// TIA Portal V16 export
// export: Created 2024-03-27T10:00:42.5235415Z, ExportSetting WithDefaults, DisplayName Totally Integrated Automation Portal, DisplayVersion V16, DisplayName TIA Portal Version Control Interface, DisplayVersion V16, DisplayName TIA Portal Openness, DisplayVersion V16, DisplayName STEP 7 Professional, DisplayVersion V16, DisplayName STEP 7 Safety, DisplayVersion V16, DisplayName WinCC Advanced, DisplayVersion V16
TYPE "UR_1_T2O_State"
// stored: IsFailsafeCompliant false
   STRUCT
      Robot { S7_SetPoint := 'True'} : "UR__T2O_Robot";
      Safety { S7_SetPoint := 'True'} : "UR__T2O_Safety";
   END_STRUCT;
END_TYPE
